// TIA Portal project "EX_DIV" (V18)

(* hardware
DEVICE "S7-1500/ET200MP station_1"  S7-1500 station
   slot 0: "Rail_0"  Rack  6ES7 590-1***0-0AA0
   slot 1: "PLC_1"  CPU 1511-1 PN  6ES7 511-1AL03-0AB0  V3.0
      slot 3: "CPU display_1"  6ES7591-1AA00-0AA0
      slot 32768: "PROFINET interface_1"  X1
         slot 32769: "Port_1"  X1 P1
         slot 32770: "Port_2"  X1 P2
      slot 34817: "Virtual CP interface port_1"  Virtual CP interface port  Virtual CP interface port
*)

// ===== PLC "PLC_1"  CPU 1511-1 PN =====

VAR_GLOBAL   // PLC tag table "Default tag table"
   "Tag_1" AT %MW1 : Int;
   "Tag_2" AT %QW1 : Word;
END_VAR

DATA_BLOCK "Data_block_1"   // DB1
{ S7_Optimized_Access := 'TRUE' }
VERSION : 0.1
   VAR
      "A" : Real;
      "B" : Real;
      Resultado : Real;
   END_VAR
BEGIN
END_DATA_BLOCK

FUNCTION "DIVISAO" : Void   // FC1, SCL
{ S7_Optimized_Access := 'TRUE' }
VERSION : 0.1
   VAR_INPUT
      "A" : Real;
      "B" : Real;
   END_VAR
   VAR_OUTPUT
      C : Real;
   END_VAR
BEGIN
   REGION MULTIPLICACAO
       #C := #A / #B;

   END_REGION
END_FUNCTION

ORGANIZATION_BLOCK "Main"   // OB1, LAD, ProgramCycle
TITLE = "Main Program Sweep (Cycle)"
{ S7_Optimized_Access := 'TRUE' }
VERSION : 0.1
   VAR_INPUT
      Initial_Call : Bool;   // Initial call of this OB
      Remanence : Bool;   // =True, if remanent data are available
   END_VAR
BEGIN

REGION Network 1
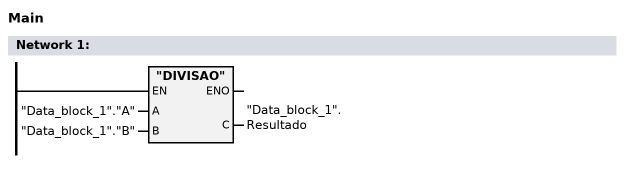
   RUNG wire#powerrail
      "DIVISAO"("A" := "Data_block_1"."A", "B" := "Data_block_1"."B", C => "Data_block_1".Resultado)
   END_RUNG
   // the same network as SCL:
   "DIVISAO"("A" := "Data_block_1"."A", "B" := "Data_block_1"."B", C => "Data_block_1".Resultado);
END_REGION
END_ORGANIZATION_BLOCK